(* IEC 61131-3 sources: atn/, 3 files *)

(* ---- atn.typ ---- *)
(*/********************************************************************
 * COPYRIGHT -- Loupe
 ********************************************************************
 * Library: All Together Now -atn
 * Author: Josh Polansky
 * Created: April 7, 2020
 ********************************************************************
 * Implementation of library All Together now
 ********************************************************************/*)

TYPE
	ATN_SST_enum :
		(
		ATN_SS_INIT (*0*)
		);
	ATN_ST_enum :
		(
		ATN_IDLE, (*0*)
		ATN_EXECUTE,
		ATN_WAITING,
		ATN_DONE,
		ATN_ABORT,
		ATN_ERROR,
		ATN_BYPASSED
		);
	ATN_ERROR_enum :
		(
		ATN_ERROR_OK := 0,
		ATN_ERROR_ACTIVE,
		ATN_ERROR_ABORTED,
		ATN_ERROR_ACTIONS_FULL,
		ATN_ERROR_BUSY := 65535
		);
	ATN_RESPONSE_ST :
		(
		ATN_RESPONSE_ST_NONE,
		ATN_RESPONSE_ST_ERROR,
		ATN_RESPONSE_ST_STEP_DONE,
		ATN_RESPONSE_ST_NEXT_STEP,
		ATN_RESPONSE_ST_STATE_DONE,
		ATN_RESPONSE_ST_BUSY
		);
	Atn_typ : 	STRUCT
		in : AtnIn_typ;
		out : AtnOut_typ;
		internal : AtnInternal_typ;
	END_STRUCT;
	AtnIn_typ : 	STRUCT
		cmd : AtnInCmd_typ;
		par : AtnInPar_typ;
	END_STRUCT;
	AtnInCmd_typ : 	STRUCT
		abort : BOOL;
		forceQuit : BOOL;
	END_STRUCT;
	AtnInPar_typ : 	STRUCT
		category : STRING[ATN_NAMESPACE_LEN];
		ID : USINT;
	END_STRUCT;
	AtnOut_typ : 	STRUCT
		activeThreads : ARRAY[0..MAI_ATN_ACT_THREADS]OF AtnActiveThread_typ;
		busy : BOOL;
		done : BOOL;
		error : BOOL;
	END_STRUCT;
	AtnOutStatus_typ : 	STRUCT
		blocked : BOOL;
		busy : BOOL;
		done : BOOL;
		error : BOOL;
	END_STRUCT;
	AtnApiStatusLocal_typ : 	STRUCT
		active : BOOL;
		busy : BOOL;
		done : BOOL;
		aborted : BOOL;
		error : BOOL;
		errorID : UDINT;
		remote : AtnApiStatus_typ;
	END_STRUCT;
	AtnApiStatus_typ : 	STRUCT
		active : BOOL;
		busy : BOOL;
		done : BOOL;
		aborted : BOOL;
		error : BOOL;
		errorID : UDINT;
	END_STRUCT;
	AtnInternal_typ : 	STRUCT
		thread : AtnThread_typ;
	END_STRUCT;
	AtnActiveThread_typ : 	STRUCT
		action : STRING[ATN_ACTION_NAME_LEN];
		busyModule : ARRAY[0..MAI_ATN_ACT_ACTIONS]OF UDINT;
		errorModule : ARRAY[0..MAI_ATN_ACT_ACTIONS]OF UDINT;
		status : AtnOutStatus_typ;
	END_STRUCT;
	AtnThread_typ : 	STRUCT
		ID : USINT;
		request : AtnActionCmdData_typ;
		activeRequest : AtnActionCmdData_typ;
		state : ATN_ST_enum;
		substate : UDINT;
		nextSubState : UDINT;
		abort : BOOL;
		forceQuit : BOOL;
		responseStatus : ATN_RESPONSE_ST;
		actions : UDINT;
		actionCount : UDINT;
		substateRequestModule : UDINT;
		busyModule : ARRAY[0..MAI_ATN_ACT_ACTIONS]OF UDINT;
		blockingModule : ARRAY[0..MAI_ATN_ACT_ACTIONS]OF UDINT;
		errorModule : ARRAY[0..MAI_ATN_ACT_ACTIONS]OF UDINT;
		activeActions : ARRAY[0..MAI_ATN_ACT_ACTIONS]OF UDINT;
		status : AtnOutStatus_typ;
	END_STRUCT;
	AtnAPI_typ : 	STRUCT
		moduleName : STRING[80];
		moduleStatus : STRING[80];
		request : STRING[ATN_ACTION_NAME_LEN];
		state : ATN_ST_enum;
		response : ATN_ST_enum;
		subState : UDINT;
		subStateReq : UDINT;
		oneShot : BOOL;
		moduleBypass : BOOL;
		moduleIsBypassed : BOOL;
		activeThread : REFERENCE TO UDINT;
		waitingThread : REFERENCE TO UDINT;
		waitingDirectorID : USINT;
	END_STRUCT;
	AtnAPIState_typ : 	STRUCT
		moduleName : STRING[80];
		moduleStatus : STRING[80];
		moduleBypass : BOOL;
		moduleIsBypassed : BOOL;
		active : BOOL;
	END_STRUCT;
	AtnActionList_typ : 	STRUCT
		name : STRING[ATN_NAMESPACE_LEN];
		maxActions : UDINT;
		pActions : REFERENCE TO AtnActionData_typ;
	END_STRUCT;
	AtnActionData_typ : 	STRUCT
		name : STRING[ATN_ACTION_NAME_LEN];
		pParameters : UDINT;
		sParameters : UDINT;
		pAction : REFERENCE TO AtnAPI_typ;
	END_STRUCT;
	AtnActionCmdData_typ : 	STRUCT
		name : STRING[ATN_ACTION_NAME_LEN];
		pParameters : UDINT;
		sParameters : UDINT;
		pStatusStructure : UDINT;
	END_STRUCT;
	AtnPlcOpenCall : 	STRUCT
		abort : BOOL;
	END_STRUCT;
	AtnPlcOpenStatus : 	STRUCT
		activeCommand : STRING[80];
		status : DINT;
		parametersWritten : BOOL;
		bypass : BOOL;
		internal : AtnPlcOpenInternal;
	END_STRUCT;
	AtnPlcOpenInternal : 	STRUCT
		fbk : UDINT;
		trig : BOOL;
	END_STRUCT;
	ATN_PLCOPEN_FUB_STATE_enum :
		(
		ATN_PLCOPEN_FUB_IDLE,
		ATN_PLCOPEN_FUB_NEW_COMMAND,
		ATN_PLCOPEN_FUB_ABORT_OLD,
		ATN_PLCOPEN_FUB_WRITE_PAR,
		ATN_PLCOPEN_FUB_SET_COMMAND,
		ATN_PLCOPEN_FUB_WORKING,
		ATN_PLCOPEN_FUB_STATUS,
		ATN_PLCOPEN_FUB_CLEANUP,
		ATN_PLCOPEN_FUB_DONE,
		ATN_PLCOPEN_FUB_ABORTED
		);
END_TYPE

(* ---- atn.fun ---- *)
(*/********************************************************************
 * COPYRIGHT -- Loupe
 ********************************************************************
 * Library: All Together Now -atn
 * Author: Josh Polansky
 * Created: April 7, 2020
 ********************************************************************
 * Implementation of library All Together now
 ********************************************************************/*)

FUNCTION atninit : UDINT
	VAR_INPUT
		buff : UDINT;
		bufsize : UDINT;
	END_VAR
END_FUNCTION

FUNCTION atncyclic : UDINT
	VAR_INPUT
		buff : UDINT;
		bufsize : UDINT;
	END_VAR
END_FUNCTION

FUNCTION_BLOCK AtnRunAction
	VAR_INPUT
		execute : BOOL;
		director : {REDUND_UNREPLICABLE} UDINT;
		action : {REDUND_UNREPLICABLE} STRING[ATN_ACTION_NAME_LEN];
		pParameters : {REDUND_UNREPLICABLE} UDINT;
		parameterSize : {REDUND_UNREPLICABLE} UDINT;
	END_VAR
	VAR_OUTPUT
		busy : BOOL;
		done : BOOL;
		active : BOOL;
		aborted : BOOL;
		error : BOOL;
	END_VAR
	VAR
		status : AtnApiStatus_typ;
		_execute : BOOL;
	END_VAR
END_FUNCTION_BLOCK
(*
Actions interface
*)

FUNCTION atnRunAction : USINT
	VAR_INPUT
		director : Atn_typ;
		action : STRING[ATN_ACTION_NAME_LEN];
		pParameters : REFERENCE TO UDINT;
		parameterSize : UDINT;
		status : AtnApiStatus_typ;
	END_VAR
END_FUNCTION

FUNCTION atnCyclic : USINT
	VAR_INPUT
		director : Atn_typ;
	END_VAR
END_FUNCTION

FUNCTION atnRegisterActionPV : USINT
	VAR_INPUT
		category : STRING[ATN_NAMESPACE_LEN];
		name : STRING[ATN_ACTION_NAME_LEN];
		actionPv : STRING[80];
		parameterPv : STRING[80];
	END_VAR
END_FUNCTION

FUNCTION atnRegisterActionPVLocal : USINT
	VAR_INPUT
		category : STRING[ATN_NAMESPACE_LEN];
		name : STRING[ATN_ACTION_NAME_LEN];
		actionPv : STRING[80];
		parameterPv : STRING[80];
	END_VAR
END_FUNCTION

FUNCTION atnRegisterAction : USINT
	VAR_INPUT
		category : STRING[ATN_NAMESPACE_LEN];
		name : STRING[ATN_ACTION_NAME_LEN];
		pAction : AtnAPI_typ;
		pParameters : REFERENCE TO UDINT;
		parameterSize : UDINT;
	END_VAR
END_FUNCTION

FUNCTION atnGetActionList : UDINT
	VAR_INPUT
		gategory : STRING[ATN_NAMESPACE_LEN];
	END_VAR
END_FUNCTION

FUNCTION atnSetActionList : BOOL
	VAR_INPUT
		gategory : STRING[ATN_NAMESPACE_LEN];
		pActions : AtnActionData_typ;
		size : UDINT;
	END_VAR
END_FUNCTION

FUNCTION populateActionList : BOOL
	VAR_INPUT
		listname : STRING[80];
	END_VAR
END_FUNCTION
(*
State/Command Interface
*)
(*Registering*)

FUNCTION registerStateBool : UDINT
	VAR_INPUT
		state : STRING[80];
		moduleName : STRING[80];
	END_VAR
	VAR_IN_OUT
		value : BOOL;
	END_VAR
END_FUNCTION

FUNCTION registerStateBoolAdr : UDINT
	VAR_INPUT
		state : STRING[80];
		moduleName : STRING[80];
		value : REFERENCE TO BOOL;
	END_VAR
END_FUNCTION

FUNCTION registerStateParameters : UDINT
	VAR_INPUT
		state : STRING[80];
		moduleName : STRING[80];
		pParameters : REFERENCE TO UDINT;
		sParameters : UDINT;
	END_VAR
END_FUNCTION

FUNCTION registerStateExt1 : UDINT
	VAR_INPUT
		state : STRING[80];
		moduleName : STRING[80];
		pModuleStatus : STRING[80];
		pParameters : REFERENCE TO UDINT;
		sParameters : UDINT;
	END_VAR
	VAR_IN_OUT
		pModuleByPass : BOOL;
		pActive : BOOL;
	END_VAR
END_FUNCTION

FUNCTION registerToResource : UDINT
	VAR_INPUT
		resource : STRING[80];
		moduleName : STRING[80];
	END_VAR
	VAR_IN_OUT
		pResourceUserId : UDINT;
		pResourceActive : BOOL;
	END_VAR
END_FUNCTION
(*Subscribing*)

FUNCTION subscribeCommandBool : UDINT
	VAR_INPUT
		commandName : STRING[80];
		moduleName : STRING[80];
	END_VAR
	VAR_IN_OUT
		command : BOOL;
	END_VAR
END_FUNCTION

FUNCTION subscribePLCOpen : UDINT
	VAR_INPUT
		commandName : STRING[80];
		moduleName : STRING[80];
	END_VAR
	VAR_IN_OUT
		command : BOOL;
		status : AtnPlcOpenStatus;
	END_VAR
END_FUNCTION

FUNCTION subscribePLCOpenWithParameters : UDINT
	VAR_INPUT
		commandName : STRING[80];
		moduleName : STRING[80];
		pParameters : REFERENCE TO UDINT;
		sParameters : UDINT;
	END_VAR
	VAR_IN_OUT
		command : BOOL;
		status : AtnPlcOpenStatus;
	END_VAR
END_FUNCTION
(*PLCOpen*)

FUNCTION atnPLCOpenAbort : BOOL
	VAR_IN_OUT
		status : AtnPlcOpenStatus;
	END_VAR
END_FUNCTION
(*
Combined State check
*)

FUNCTION stateAllTrue : BOOL
	VAR_INPUT
		state : STRING[80];
		fallback : BOOL;
	END_VAR
END_FUNCTION

FUNCTION stateAnyTrue : BOOL
	VAR_INPUT
		state : STRING[80];
		fallback : BOOL;
	END_VAR
END_FUNCTION

FUNCTION stateAllFalse : BOOL
	VAR_INPUT
		state : STRING[80];
		fallback : BOOL;
	END_VAR
END_FUNCTION

FUNCTION stateAnyFalse : BOOL
	VAR_INPUT
		state : STRING[80];
		fallback : BOOL;
	END_VAR
END_FUNCTION

FUNCTION_BLOCK stateAllTrueFb
	VAR_INPUT
		update : BOOL;
		state : {REDUND_UNREPLICABLE} STRING[80];
		fallback : {REDUND_UNREPLICABLE} BOOL;
	END_VAR
	VAR_OUTPUT
		value : BOOL;
	END_VAR
	VAR
		cache : REFERENCE TO UDINT;
	END_VAR
END_FUNCTION_BLOCK

FUNCTION_BLOCK stateAnyTrueFb
	VAR_INPUT
		update : BOOL;
		state : {REDUND_UNREPLICABLE} STRING[80];
		fallback : {REDUND_UNREPLICABLE} BOOL;
	END_VAR
	VAR_OUTPUT
		value : BOOL;
	END_VAR
	VAR
		cache : REFERENCE TO UDINT;
	END_VAR
END_FUNCTION_BLOCK

FUNCTION_BLOCK stateAllFalseFb
	VAR_INPUT
		update : BOOL;
		state : {REDUND_UNREPLICABLE} STRING[80];
		fallback : {REDUND_UNREPLICABLE} BOOL;
	END_VAR
	VAR_OUTPUT
		value : BOOL;
	END_VAR
	VAR
		cache : REFERENCE TO UDINT;
	END_VAR
END_FUNCTION_BLOCK

FUNCTION_BLOCK stateAnyFalseFb
	VAR_INPUT
		update : BOOL;
		state : {REDUND_UNREPLICABLE} STRING[80];
		fallback : {REDUND_UNREPLICABLE} BOOL;
	END_VAR
	VAR_OUTPUT
		value : BOOL;
	END_VAR
	VAR
		cache : REFERENCE TO UDINT;
	END_VAR
END_FUNCTION_BLOCK
(*
Individual State check
*)

FUNCTION stateCount : INT
	VAR_INPUT
		State : STRING[80];
	END_VAR
END_FUNCTION

FUNCTION forState : BOOL
	VAR_INPUT
		State : STRING[80];
		indexer : INT;
		active : REFERENCE TO BOOL;
		pParameters : REFERENCE TO UDINT;
		sParameters : UDINT;
	END_VAR
END_FUNCTION

FUNCTION forStateGetPointer : BOOL
	VAR_INPUT
		State : STRING[80];
		indexer : INT;
		active : REFERENCE TO BOOL;
		pParameters : REFERENCE TO UDINT;
		sParameters : REFERENCE TO UDINT;
	END_VAR
END_FUNCTION
(*
Executing Commands*)

FUNCTION executeCommand : BOOL
	VAR_INPUT
		Command : STRING[80];
	END_VAR
END_FUNCTION

FUNCTION_BLOCK AtnPLCOpen
	VAR_INPUT
		Command : STRING[80];
		Execute : BOOL;
		Fallback : DINT;
	END_VAR
	VAR_OUTPUT
		Status : DINT;
		StatusMessage : ARRAY[0..9] OF STRING[80];
		Busy : BOOL;
		Done : BOOL;
		Aborted : BOOL;
		Error : BOOL;
	END_VAR
	VAR
		_state : USINT;
		_command : {REDUND_UNREPLICABLE} UDINT;
		_execute : BOOL;
		_call : AtnPlcOpenCall;
	END_VAR
END_FUNCTION_BLOCK

FUNCTION_BLOCK AtnPLCOpenWithParameters
	VAR_INPUT
		Command : STRING[80];
		Execute : BOOL;
		Fallback : DINT;
		pParameters : REFERENCE TO UDINT;
		sParameters : {REDUND_UNREPLICABLE} UDINT;
	END_VAR
	VAR_OUTPUT
		Status : DINT;
		StatusMessage : ARRAY[0..9] OF STRING[80];
		Busy : BOOL;
		Done : BOOL;
		Aborted : BOOL;
		Error : BOOL;
	END_VAR
	VAR
		_state : USINT;
		_command : {REDUND_UNREPLICABLE} UDINT;
		_execute : BOOL;
		_call : AtnPlcOpenCall;
	END_VAR
END_FUNCTION_BLOCK
(*Reading Status*)

FUNCTION stateTrueStatus : BOOL
	VAR_INPUT
		state : STRING[80];
		buffer : UDINT;
		sBuffer : UDINT;
	END_VAR
END_FUNCTION

FUNCTION stateFalseStatus : BOOL
	VAR_INPUT
		state : STRING[80];
		buffer : UDINT;
		sBuffer : UDINT;
	END_VAR
END_FUNCTION

FUNCTION stateStatus : BOOL
	VAR_INPUT
		state : STRING[80];
		buffer : UDINT;
		sBuffer : UDINT;
	END_VAR
END_FUNCTION

FUNCTION systemJson : BOOL
	VAR_INPUT
		buffer : UDINT;
		sBuffer : UDINT;
	END_VAR
END_FUNCTION
(*Application Functions*)

FUNCTION resourceIsAvailable : BOOL
	VAR_INPUT
		resourceName : STRING[80];
		resourceUserId : UDINT;
	END_VAR
END_FUNCTION

FUNCTION isInhibited : BOOL
	VAR_INPUT
		inhibit : STRING[80];
	END_VAR
END_FUNCTION

(* ---- atn.var ---- *)
(*/********************************************************************
 * COPYRIGHT -- Loupe
 ********************************************************************
 * Library: All Together Now -atn
 * Author: Josh Polansky
 * Created: April 7, 2020
 ********************************************************************
 * Implementation of library All Together now
 ********************************************************************/*)
VAR CONSTANT
	MAI_ATN_ACTIONS : USINT := 99;
	MAI_ATN_ACTIONLISTS : USINT := 9;
	MAI_ATN_ACT_ACTIONS : USINT := 10;
	MAI_ATN_ACT_THREADS : USINT := 0;
	ATN_ACTION_NAME_LEN : USINT := 20;
	ATN_NAMESPACE_LEN : USINT := 20;
END_VAR
